FUNCTION_BLOCK FB_GUI_TEST
VAR_INPUT
	iLevel :INT;
	nCount: INT:=0;
END_VAR
VAR
	bInitialise : BOOL := FALSE;
	bStartCycle : BOOL := FALSE;
	tCaptureDelay: TIME:= T#1000MS;
	tDelayNextStep: TIME:= T#200MS;
	tInterval: TIME:= T#250MS;
	
	bCylinderUp : BOOL;
	//iLevel : UINT :=2; 
	
	nState : UINT :=0;
	//nCount: INT:=0;
	nNoOfCycle:INT:=1;
	TDelay : TON;
	TDelay1 : TON;
	bUp: BOOL;
	sErr: STRING;
	tempstr : ARRAY[1..4] OF STRING;
	tempstrRet : ARRAY[1..4] OF STRING;
	str: STRING;
	TDelay2 : TON;
	i: INT :=1;
	
	bCylinderOutL1: BOOL;
	bOutL1 : BOOL;
	
	bPBStart : BOOL;
	
	StartPbDly: TON;
	rtStartTrig :R_Trig;
	
	
	iClearCount: INT;
	iTotalClear: INT:=20;
	ClearTCSEvent: TON;
	mlVIO:ST_TCMultiLevel_VIO; 
END_VAR
VAR_IN_OUT
	bStart:BOOL;
END_VAR

IF bInitialise THEN
	arrTCMultiLevel[iLevel].stGblParam.bInitialise:=TRUE;
	bInitialise:=FALSE;
END_IF

IF bCylinderUp THEN
	IF (arrTCMultiLevel[iLevel].fbTCMultiLevelSeq.M_nCmptUpDown(bUp, sErr)=10) THEN
		bCylinderUp :=FALSE;
	END_IF
END_IF

IF bCylinderOutL1 THEN
	IF (arrTCMultiLevel[iLevel].fbTCMultiLevelSeq.M_nCmptInOut(bOutL1, sErr)=10) THEN
		bCylinderOutL1 :=FALSE;
	END_IF
END_IF

(*StartPbDly(in:=(stIO[iLevel].ipStartPB),pt:=T#100MS);
rtStartTrig(Clk:=StartPbDly.Q);
IF rtStartTrig.Q THEN
	bPBStart:=TRUE;
END_IF *)

bPBStart := arrTCVIO[iLevel].ipStartPB;

IF bStartCycle XOR bStart THEN //cycle Up down, in out
	CASE nState OF
		0: //Out
	 		TDelay(IN:=FALSE);
	 		TDelay1(IN:=FALSE);
			TDelay2(IN:=FALSE);
			i:=1;
			nState := 1;
		1: //Out
	 		//TDelay(IN:=FALSE);
	 		//TDelay1(IN:=FALSE);
			//TDelay2(IN:=FALSE);
			//i:=1;
			//arrTCMultiLevel[iLevel].stGblParam.bShuttleMoveOut := TRUE;
			//<MoveOut>
				arrTACommands.arrTACommands[1].sLogName := CONCAT('TIUSlideOut_TESTER_LA',CONCAT('0',INT_TO_STRING(iLevel)));
				arrTACommands.arrTACommands[1].eTaskName := E_TaskName.TIUSlideOut;
				arrTACommands.arrTACommands[1].eModuleID := LevelModuleID[iLevel];
				arrTACommands.arrTACommands[1].bParam[1] := TRUE;
				arrTCSCommandReady:= FALSE;
				iClearCount := iTotalClear;
				
				ClearTCSEvent(IN:=(iClearCount > 0), PT:=T#100MS);
				IF ClearTCSEvent.Q THEN
					ClearTCSEvent(IN:=FALSE);
					iClearCount := iClearCount - 1;
					arrTCSEventTriggered:= FALSE;
				END_IF
			//</region>
			
	 		nState := 2;
	 2:		mlVIO:= arrTCMultiLevel[iLevel].fbTCMultiLevelSeq.P_stTCMultiLevelVIO;
			IF mlVIO.ipTCDrawerCylExtendRS= TRUE THEN
	 			nState := 3;
			END_IF
	 //Delay					
	 3: 	IF arrTCMultiLevel[iLevel].stGblParam.bShuttleMoveOut =FALSE THEN
		    	IF iLevel = 3 THEN   // Level No for Distance Laser Sensor Reading
		 			TDelay1(IN:=TRUE,PT:=tCaptureDelay);
					IF TDelay1.Q THEN
						TDelay2(IN:=TRUE,PT:=tInterval);
						IF TDelay2.Q THEN			
							TDelay2(IN:=FALSE);
							tempstr[1] := F_concat3('XE,', REAL_TO_STRING(aiXConverted[iLevel]), ', ');
							tempstr[2] := F_concat3('YE,', REAL_TO_STRING(aiYConverted[iLevel]), ', ');
							tempstr[3] := F_concat3('ZE,', REAL_TO_STRING(aiZConverted[iLevel]), ', ');
							tempstr[4] := F_concat3(tempstr[1], tempstr[2], tempstr[3]);
							
							tempstrRet[1] := F_concat3('XR,', REAL_TO_STRING(aiXConvertedRet[iLevel]), ', ');
							tempstrRet[2] := F_concat3('YR,', REAL_TO_STRING(aiYConvertedRet[iLevel]), ', ');
							tempstrRet[3] := F_concat3('ZR,', REAL_TO_STRING(aiZConvertedRet[iLevel]), ', ');
							tempstrRet[4] := F_concat3(tempstrRet[1], tempstrRet[2], tempstrRet[3]);
							
							str:= '';
							str:= CONCAT(tempstr[4] , tempstrRet[4]);
							Logging.fbDebugLog.M_nLogger(1, sSource:='aisensor', F_concat3(INT_TO_STRING(i), ', ', str));
							
							//Logging.fbDebugLog.M_nLogger(1, sSource:='aisensor', F_concat3(INT_TO_STRING(i), ', ', tempstr[4]));
							i := i+1;
							IF i>4 THEN
								nState := 4;
							END_IF
						END_IF
						//END_FOR
					END_IF
					(*
					TDelay(IN:=TRUE,PT:=tDelayNextStep);//after move out, delay before move in
					IF TDelay.Q THEN
						TDelay(IN:=FALSE);
						nState := 3;
					END_IF
					*)
					
				ELSE
					nState := 4;
				END_IF
				
			END_IF

	 4:		//In
			//arrTCMultiLevel[iLevel].stGblParam.bShuttleMoveIn := TRUE;
	 		//<MoveIn>
				arrTACommands.arrTACommands[1].sLogName := CONCAT('TIUSlideOut_TESTER_LA',CONCAT('0',INT_TO_STRING(iLevel)));
				arrTACommands.arrTACommands[1].eTaskName := E_TaskName.TIUSlideOut;
				arrTACommands.arrTACommands[1].eModuleID := LevelModuleID[iLevel];
				arrTACommands.arrTACommands[1].bParam[1] := FALSE;
				arrTCSCommandReady:= FALSE;
				iClearCount := iTotalClear;
				
				ClearTCSEvent(IN:=(iClearCount > 0), PT:=T#100MS);
				IF ClearTCSEvent.Q THEN
					ClearTCSEvent(IN:=FALSE);
					iClearCount := iClearCount - 1;
					arrTCSEventTriggered:= FALSE;
				END_IF
			//</MoveIn>
			
	 		nState := 5;
			
	5:
	 		mlVIO:= arrTCMultiLevel[iLevel].fbTCMultiLevelSeq.P_stTCMultiLevelVIO;
			IF mlVIO.ipTCDrawerCylRetractRS= TRUE THEN
	 			nState := 6;
			END_IF
			//Done
	 6: 	IF arrTCMultiLevel[iLevel].stGblParam.bShuttleMoveIn=FALSE THEN
			TDelay(IN:=TRUE,PT:=tDelayNextStep);//after move out, delay before move in
			IF TDelay.Q THEN
				TDelay(IN:=FALSE);
				nState := 0;
				nCount := nCount +1;
			END_IF	 
	 
			END_IF
	END_CASE
	
	IF nCount> nNoOfCycle(*AND nState =3*) THEN
		bStartCycle := FALSE;
		bStart:=FALSE;
		nCount:=1;
		//bPBStart := FALSE;
		
	END_IF
		
END_IF

END_FUNCTION_BLOCK

(* stored: Version 1.1.0.1, ProductVersion 3.1.4022.18
   POU FB_GUI_TEST: Id {2d2d503a-f036-4331-9480-856b87027775}, SpecialFunc None *)
